(* PLC project Generated.project, CODESYS CODESYS V3.5 SP19 Patch 1 *)
(* stored: creationDateTime 2026-09-06T13:00:42.501848, modificationDateTime 2026-09-06T13:00:42.501848 *)

TYPE ST_Chain_Translation_Safety : STRUCT
  Idx301_EmergencyChainClosed : BOOL;  (* 1 = Boucle Urgence OK | 0 = Arrêt d'Urgence Appuyé *)
  Idx302_SafeStopActive : BOOL;  (* 0 = Sain (Autorisé) | 1 = Arrêt Rapide Translation *)
  Idx303_PowerCutOffActive : BOOL;  (* 0 = Puissance OK | 1 = Coupure Puissance *)
  Idx304_LimitSwitchTremieActive : BOOL;  (* 0 = Sain | 1 = Fin de Course Extrême Trémie (ex-Idx304_LimitSwitchFwdActive) *)
  Idx305_LimitSwitchMaintenanceActive : BOOL;  (* 0 = Sain | 1 = Fin de Course Extrême Maintenance (ex-Idx305_LimitSwitchRevActive) *)
  Idx306_BypassLimitSwitch : BOOL;  (* 0 = Fins de course actives | 1 = Shuntés IHM ⚠️ *)
  Idx307_PositionDecoderIncoherent : BOOL;  (* 0 = Décodage 5 Capteurs OK | 1 = Incohérence Position *)
  Idx308_HeightInterlockBlocking : BOOL;  (* : 0 = M1 ET M2 ≥ hauteur mini (ou bypass) | 1 = Translation bloquée (risque collision) *)
  Idx309_ErrorOperatorComm : BOOL;  (* Défauts safety déchiffrés (bits ErrorId) — visibles individuellement à l'IHM bit0 Perte communication opérateur (joystick CAN / heartbeat IHM) *)
  Idx310_ErrorDriveComm : BOOL;  (* bit1 Perte communication EtherCAT variateur *)
  Idx311_ErrorPhaseRotation : BOOL;  (* bit2 Mauvaise rotation de phases *)
  Idx312_ErrorBrakeThermal : BOOL;  (* bit3 Surchauffe thermique frein commun *)
  Idx313_ErrorMecaB : BOOL;  (* bit4 Absence confirmation arrêt *)
  Idx314_ErrorMecaA : BOOL;  (* bit5 Mouvement non commandé *)
  Idx315_ErrorLimitSwitch : BOOL;  (* bit6 Limite extrême atteinte *)
  Idx316_ErrorSensorIncoherent : BOOL;  (* bit7 Mot capteurs position incohérent *)
  Idx317_ErrorId : WORD;  (* Masque brut complet (latch cause) — source d'arbitrage PowerCutOff *)
  Idx318_EffectivePermitM3_Tremie : BOOL;  (* Permis directionnels M3 (source unique : FB_Safety_Translation) — TRUE = autorisé, fail-safe 1 = Translation vers Trémie autorisée | 0 = SENS TRÉMIE BLOQUÉ *)
  Idx319_EffectivePermitM3_Maintenance : BOOL;  (* 1 = Translation vers Maintenance/P1 autorisée | 0 = SENS MAINTENANCE BLOQUÉ *)
END_STRUCT;
END_TYPE
